# B&R Automation Studio project AutomationsProject
Automation Studio 4.12.6.106; technology packages: mappMotion 5.30.2, mappView 5.24.7

## Configuration Config1

CPU X20CP1382, AutomationRuntime I4.83, Build 4.1.2, Vc V4.73.2

### Task classes (Cpu.sw)
```
Cyclic#4:
  RunBelt <- RunBelt.prg
  main <- main.prg
  ServoTest <- ServoTest.prg
DataObjects: McAcpSys
NcDataObjects: mcdrivelog
Binaries: FWRules, udbdef, TCData, McAcpSim, McAcpDrv, arconfig, User, sysconf, Role, iomap, asfw, ashwac, ashwd, Config_1, arcoal, arsvcreg, arflatprv
Libraries: CppLibs, McBase, MpBase, McAxis, MpAxis, McAcpAx, astime, asieccon, fileio, runtime, powerlnk, asepl, sys_lib
```

### Hardware
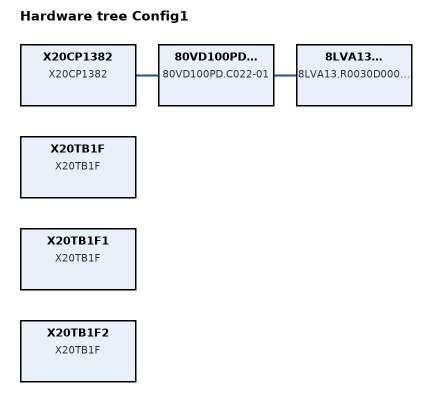
```
80VD100PD.C022-01 : 80VD100PD.C022-01 v2.5.0.0  [PLK1 -> X20CP1382.IF3 (NodeNumber=1) [Cable Type=PowerlinkCable, Length=10, Version=1.0.0.3]; EC1 -> 8LVA13.R0030D000-0.EC]
  DriveConfiguration/Module:
    McAcoposTypeID = AcoposMicroDConfig
    ActivateACOPOSSimulationOnPLC = 0
  DriveConfiguration/Encoder/EncoderX6A/InterfaceType:
    ResolverPolepairs = 1
  DriveConfiguration/Encoder/EncoderX6B/InterfaceType:
    ResolverPolepairs = 1
  DriveConfiguration/Channel[1]/RealAxis:
    AxisReference = FeederAxis
    MechanicalElementsIsInvisible = 0
  DriveConfiguration/Channel[1]/RealAxis/MechanicalElements/Gearbox:
    InputIsReadOnly = 0
    Input = 1
    OutputIsReadOnly = 0
    Output = 1
  DriveConfiguration/Channel[1]/RealAxis/MechanicalElements/RotaryToLinearTransformation:
    ReferenceDistanceIsReadOnly = 0
    ReferenceDistance = 1
  DriveConfiguration/Channel[1]/RealAxis/Controller:
    ModeIsReadOnly = 0
    Mode = PositionController
  DriveConfiguration/Channel[1]/RealAxis/Controller/Mode/Position:
    ProportionalGain = 50
    IntegrationTime = 0.0
    PredictionTime = 0.0004
    TotalDelayTime = 0.0004
  DriveConfiguration/Channel[1]/RealAxis/Controller/Mode/Speed:
    ProportionalGainIsReadOnly = 0
    ProportionalGain = 0.5
    IntegrationTimeIsReadOnly = 0
    IntegrationTime = 0.0
    FilterTimeIsReadOnly = 0
    FilterTime = 0.0
  DriveConfiguration/Channel[1]/RealAxis/Controller/Mode/LoopFilters:
    LoopFilterXIsReadOnly = 0
    LoopFilter1 = NotUsed
    LoopFilter2 = NotUsed
    LoopFilter3 = NotUsed
  DriveConfiguration/Channel[1]/RealAxis/Homing:
    ModeIsReadOnly = 0
    Mode = Direct
  DriveConfiguration/Channel[1]/RealAxis/Homing/Mode:
    Position = 0.0
    ReferencePulse = NotUsed
  DriveConfiguration/Channel[1]/RealAxis/Homing:
    RestorePositionVariable = 
  DriveConfiguration/Channel[1]/RealAxis/StopReaction:
    QuickstopIsReadOnly = 0
    Quickstop = DecelerationLimit
    DriveErrorIsReadOnly = 0
    DriveError = DecelerationLimit
    FilterTime = 0.0
  DriveConfiguration/Channel[1]/RealAxis/MovementErrorLimits:
    PositionError = 1.0
    VelocityErrorMonitoring = NotUsed
  DriveConfiguration/Channel[1]/RealAxis:
    JerkFilterIsReadOnly = 0
    JerkFilter = NotUsed
    ZeroVibrationFilter = NotUsed
  DriveConfiguration/Channel[1]/RealAxis/DigitalInputs/HomingSwitch:
    SourceIsReadOnly = 0
    Source = NotUsed
    Level = High
  DriveConfiguration/Channel[1]/RealAxis/DigitalInputs/PositiveLimitSwitch:
    SourceIsReadOnly = 0
    Source = NotUsed
    Level = High
  DriveConfiguration/Channel[1]/RealAxis/DigitalInputs/NegativeLimitSwitch:
    SourceIsReadOnly = 0
    Source = NotUsed
    Level = High
  DriveConfiguration/Channel[1]/RealAxis/DigitalInputs/Trigger1:
    Source = X2Trigger1
    Level = High
  DriveConfiguration/Channel[1]/RealAxis/DigitalInputs/Trigger2:
    Source = X2Trigger2
    Level = High
  DriveConfiguration/Channel[1]/RealAxis/DigitalInputs/Quickstop:
    Input = Trigger2
  DriveConfiguration/Channel[1]/RealAxis/Simulation:
    SimulationModeOnPLC = SetValueGeneration
    SimulationModeOnACOPOS = NotUsed
  DriveConfiguration/Channel[1]:
    ExternalEncoderAxis = NotUsed
  DriveConfiguration/Channel[2]/RealAxis:
    AxisReference = 
    MechanicalElementsIsInvisible = 0
  DriveConfiguration/Channel[2]/RealAxis/MechanicalElements/Gearbox:
    InputIsReadOnly = 0
    Input = 1
    OutputIsReadOnly = 0
    Output = 1
  DriveConfiguration/Channel[2]/RealAxis/MechanicalElements/RotaryToLinearTransformation:
    ReferenceDistanceIsReadOnly = 0
    ReferenceDistance = 1
  DriveConfiguration/Channel[2]/RealAxis/Controller:
    ModeIsReadOnly = 0
    Mode = PositionController
  DriveConfiguration/Channel[2]/RealAxis/Controller/Mode/Position:
    ProportionalGain = 50.0
    IntegrationTime = 0.0
    PredictionTime = 0.0004
    TotalDelayTime = 0.0004
  DriveConfiguration/Channel[2]/RealAxis/Controller/Mode/Speed:
    ProportionalGainIsReadOnly = 0
    ProportionalGain = 2.0
    IntegrationTimeIsReadOnly = 0
    IntegrationTime = 0.0
    FilterTimeIsReadOnly = 0
    FilterTime = 0.0
  DriveConfiguration/Channel[2]/RealAxis/Controller/Mode/LoopFilters:
    LoopFilterXIsReadOnly = 0
    LoopFilter1 = NotUsed
    LoopFilter2 = NotUsed
    LoopFilter3 = NotUsed
  DriveConfiguration/Channel[2]/RealAxis/Homing:
    ModeIsReadOnly = 0
    Mode = Direct
  DriveConfiguration/Channel[2]/RealAxis/Homing/Mode:
    Position = 0.0
    ReferencePulse = NotUsed
  DriveConfiguration/Channel[2]/RealAxis/Homing:
    RestorePositionVariable = 
  DriveConfiguration/Channel[2]/RealAxis/StopReaction:
    QuickstopIsReadOnly = 0
    Quickstop = DecelerationLimit
    DriveErrorIsReadOnly = 0
    DriveError = DecelerationLimit
    FilterTime = 0.0
  DriveConfiguration/Channel[2]/RealAxis/MovementErrorLimits:
    PositionError = 1.0
    VelocityErrorMonitoring = Automatic1
  DriveConfiguration/Channel[2]/RealAxis:
    JerkFilterIsReadOnly = 0
    JerkFilter = NotUsed
    ZeroVibrationFilter = NotUsed
  DriveConfiguration/Channel[2]/RealAxis/DigitalInputs/HomingSwitch:
    SourceIsReadOnly = 0
    Source = NotUsed
    Level = High
  DriveConfiguration/Channel[2]/RealAxis/DigitalInputs/PositiveLimitSwitch:
    SourceIsReadOnly = 0
    Source = NotUsed
    Level = High
  DriveConfiguration/Channel[2]/RealAxis/DigitalInputs/NegativeLimitSwitch:
    SourceIsReadOnly = 0
    Source = NotUsed
    Level = High
  DriveConfiguration/Channel[2]/RealAxis/DigitalInputs/Trigger1:
    Source = X2Trigger1
    Level = High
  DriveConfiguration/Channel[2]/RealAxis/DigitalInputs/Trigger2:
    Source = X2Trigger2
    Level = High
  DriveConfiguration/Channel[2]/RealAxis/DigitalInputs/Quickstop:
    Input = Trigger2
  DriveConfiguration/Channel[2]/RealAxis/Simulation:
    SimulationModeOnPLC = SetValueGeneration
    SimulationModeOnACOPOS = NotUsed
  DriveConfiguration/Channel[2]:
    ExternalEncoderAxis = NotUsed
8LVA13.R0030D000-0 : 8LVA13.R0030D000-0 v2.2.0.5  [EC -> 80VD100PD.C022-01.EC1; MT -> 80VD100PD.C022-01.MT1]
  M1/MotorParameters:
    MOTOR_AMB_TEMP_RATED = 40
X20CP1382 : X20CP1382 v1.15.0.0  [X1 -> X1.SL; X2 -> X2.SL; X3 -> X3.SL]
  Module X1 (Type=X1, Virtual=true, Version=1.15.0.0)
    Connection (Connector=SS1, TargetModule=X20TB1F, TargetConnector=SS)
    Connection (Connector=SL, TargetModule=X20CP1382, TargetConnector=X1)
    X1AI_ChannelType01 = 4 to 20mA
  Module X2 (Type=X2, Virtual=true, Version=1.15.0.0)
    Connection (Connector=SS1, TargetModule=X20TB1F1, TargetConnector=SS)
    Connection (Connector=SL, TargetModule=X20CP1382, TargetConnector=X2)
  Module X3 (Type=X3, Virtual=true, Version=1.15.0.0)
    Connection (Connector=SS1, TargetModule=X20TB1F2, TargetConnector=SS)
    Connection (Connector=SL, TargetModule=X20CP1382, TargetConnector=X3)
    X3Channel09Source = PWMout
    X3Channel10Source = PWMout
  Connector IF2:
    ActivateDevice = 1
    Mode = Manual
    InternetAddress = 192.168.1.5
    SubnetMask = 255.255.255.0
    InaNodeNumber = 0
  ConfigurationID = testFreq_Config1
  ActivateOpcUa = 1
  OpcUaInformationModels_PV_Version = 1
X20TB1F : X20TB1F v1.0.0.0
X20TB1F1 : X20TB1F v1.0.0.0
X20TB1F2 : X20TB1F v1.0.0.0
```

### IoMap.iom - X20CP1382/IoMap.iom
```iecst
VAR_CONFIG
	::IO_Output.BELT_START AT %QX."X3".DigitalOutput01; (*24 VDC / 0.5 A, source To I1*)
	::IO_Output.BELT_DIR AT %QX."X3".DigitalOutput02; (*24 VDC / 0.5 A, source To I2*)
	::IO_Output.BELT_CONST_SPEED AT %QX."X3".DigitalOutput03; (*24 VDC / 0.5 A, source To I5*)
	::IO_Output._BELT_ACC_ AT %QW."X3".PWMOutput09; (*Pulse width modulation, 24 VDC / 0.2 A [0 to 100.0 %] To I3*)
	::IO_Output._BELT_DEACC_ AT %QW."X3".PWMOutput10; (*Pulse width modulation, 24 VDC / 0.2 A [0 to 100.0 %] To I4*)
	::IO_Output.PWM_PERIOD AT %QW."X3".PWMPeriod09;
	::IO_Output.PWM_PERIOD AT %QW."X3".PWMPeriod10;
	::IO_Input._Distance AT %IW."X1".AnalogInput01;
	::IO_Input.ROBOT_READY AT %IX."X1".DigitalInput01;
	::IO_Output.ROBOT_RUN_PRG AT %QX."X3".DigitalOutput07;
END_VAR
```

### Config_1.axis - X20CP1382/mappMotion/Config_1.axis
```
Element FeederAxis (Type=axis)
  BaseTypeIsReadOnly = 0
  BaseType = Linear
    MeasurementUnit = 5066068
    MeasurementResolutionIsReadOnly = 0
    MeasurementResolution = 0.01
    CountDirectionIsReadOnly = 0
    CountDirection = Standard
  MovementLimitsIsReadOnly = 0
  MovementLimits = Internal
    Position:
      LowerLimitMin = -1.79769313486231E308
      UpperLimitMax = 1.79769313486231E308
      LowerLimit = -1000.0
      UpperLimit = 1000.0
    VelocityIsReadOnly = 0
    Velocity:
      VelocityMax = 3.4E38
      Velocity = 10.0
    AccelerationIsReadOnly = 0
    Acceleration:
      AccelerationMax = 3.4E38
      Acceleration = 50.0
    DecelerationIsReadOnly = 0
    Deceleration:
      DecelerationMax = 3.4E38
      Deceleration = 50.0
  Alarms = None
```

## Logical view

Binary libraries used (declarations not repeated): operator, runtime, astime, AsIecCon, McBase 5.30.2, MpBase, McAxis 5.30.2, MpAxis 5.30.2, McAcpAx 5.30.2

### Global.typ - Global data types
```iecst
TYPE
	ST_Output : 	STRUCT
		PWM_PERIOD : UINT;
		BELT_START : BOOL; (*I1*)
		BELT_DIR : BOOL; (*I2*)
		BELT_CONST_SPEED : BOOL; (*I5*)
		_BELT_DEACC_ : INT; (*I4*)
		_BELT_ACC_ : INT; (*I3*)
		ROBOT_RUN_PRG : BOOL;
	END_STRUCT;
	ST_Input : 	STRUCT
		_Distance : INT; (*Distance sensor on the bottom of the track*)
		ROBOT_READY : BOOL;
		Distance : REAL;
	END_STRUCT;
	packML :
		(
		EXECUTE,
		COMPLETING,
		COMPLETED,
		RESETTING,
		ABORTING,
		ABORTED,
		CLEARING,
		STOPPING,
		STOPPED,
		SUSPENDING,
		SUSPENDED,
		UNSUSPENDING,
		UNHOLDING,
		HELD,
		HOLDING,
		STARTING,
		IDLE
		);
END_TYPE
```

### Global.var - Global variables
```iecst
VAR
	IO_Output : ST_Output;
	IO_Input : ST_Input;
END_VAR
VAR CONSTANT
	ACCEPTED_DISTANCE : REAL := 0.005;
	ROBOT_CATCH_DISTANCE : REAL := 0.22;
END_VAR
```

### Package Logical/Libraries - Global libraries

### Library Logical/Libraries/CppLibs (ANSIC)

#### myStdLib.h
```c
#ifndef MYSTDLIB_H
#define MYSTDLIB_H

#include <stdlib.h>

template<typename T>
inline T abs(T x)
{
	return x < 0 ? -x : x;
}

#endif
```

### Program Logical/main (IEC)

#### Variables.var
```iecst
VAR
	PACK_ML : packML;
	PackMLChar : STRING[80];
END_VAR
```

#### Action.st
```iecst
ACTION States:
	CASE PACK_ML OF
		ABORTING:
			PackMLChar := 'ABORTING';
			PACK_ML := ABORTED;

		ABORTED:
			PackMLChar := 'ABORTED';
			PACK_ML := CLEARING;

		CLEARING:
			PackMLChar := 'CLEARING';
			PACK_ML := STOPPED;

		STOPPING:
			PackMLChar := 'STOPPING';
			PACK_ML := ABORTED;

		STOPPED:
			PackMLChar := 'STOPPED';
			PACK_ML := RESETTING;

		RESETTING:
			PackMLChar := 'RESETTING';
			PACK_ML := IDLE;

		IDLE:
			PackMLChar := 'IDLE';
			PACK_ML := STARTING;

		STARTING:
			PackMLChar := 'STARTING';
			PACK_ML := EXECUTE;

		EXECUTE:
			PackMLChar := 'EXECUTE';
			(*

			The belt should run. If we are in an acceptable region we should go to the position of tray and catch it with the robot.
			This program only tells the robot TO run, not where TO run.

			*)
			IF ACCEPTED_DISTANCE > ABS(ROBOT_CATCH_DISTANCE - IO_Input.Distance) THEN
				IF IO_Input.ROBOT_READY THEN
					IO_Output.BELT_START := FALSE;
					IO_Output.ROBOT_RUN_PRG := TRUE;
				ELSE
					IO_Output.BELT_START := FALSE;
					IO_Output.ROBOT_RUN_PRG := FALSE;
				END_IF
			ELSE
				IO_Output.ROBOT_RUN_PRG := FALSE;

				IF (ROBOT_CATCH_DISTANCE - IO_Input.Distance) > 0 THEN
					IO_Output.BELT_CONST_SPEED := TRUE;
					IO_Output.BELT_DIR := TRUE;
					IO_Output.BELT_START := TRUE;
				ELSE
					IO_Output.BELT_CONST_SPEED := TRUE;
					IO_Output.BELT_DIR := FALSE;
					IO_Output.BELT_START := TRUE;
				END_IF

			END_IF

			//PACK_ML := COMPLETING;
		SUSPENDING:
			PackMLChar := 'SUSPENDING';
			PACK_ML := SUSPENDED;

		SUSPENDED:
			PackMLChar := 'SUSPENDED';
			PACK_ML := UNSUSPENDING;

		UNSUSPENDING:
			PackMLChar := 'UNSUSPENDING';
			PACK_ML := EXECUTE;

		HOLDING:
			PackMLChar := 'HOLDING';
			PACK_ML := HELD;

		HELD:
			PackMLChar := 'HELD';
			PACK_ML := UNHOLDING;

		UNHOLDING:
			PackMLChar := 'UNHOLDING';
			PACK_ML := EXECUTE;

		COMPLETING:
			PackMLChar := 'COMPLETING';
			PACK_ML := COMPLETED;

		COMPLETED:
			PackMLChar := 'COMPLETED';
			PACK_ML := RESETTING;

	END_CASE
END_ACTION
```

#### Main.st
```iecst
PROGRAM _INIT
	(* Insert code here *)

	PACK_ML := CLEARING;

END_PROGRAM

PROGRAM _CYCLIC
	(* Insert code here *)

	IF IO_Input._Distance < 1000 OR IO_Input._Distance > 32000 THEN
		IO_Input.Distance := 1.0;
	ELSE
		IO_Input.Distance := 0.00001033592*IO_Input._Distance+0.1581395;
	END_IF

	States;  // action

	IO_Input.ROBOT_READY; //Kanal 601 - output på robot

	IO_Output.ROBOT_RUN_PRG; //Kanal 501 - input på robot

END_PROGRAM

PROGRAM _EXIT
	(* Insert code here *)

END_PROGRAM
```

### Program Logical/RunBelt (ANSIC)

#### Variables.var
```iecst
VAR
	BELT_SPEED : REAL; (*Belt speed target*)
	_BELT_CURRENT_SPEED_ : REAL; (*Current belt speed*)
	_BELT_ACCELERATION_ : INT; (*Acceleration to belt speed target*)
END_VAR
```

#### Main.cpp
```cpp
#include <bur/plctypes.h>
#ifdef _DEFAULT_INCLUDES
	#include <AsDefault.h>
#endif

#include <cmath>
#include <string>
#include <vector>
#include <map>
#include "../Libraries/CppLibs/myStdLib.h"
//#include <myStdLib.h>

#define INDIFFERENT_SPEED_DIFF 0.5 // [m/s]

std::vector<double> something(50);

// amount of memory to be allocated for heap storage must be specified for every ANSI C++ program with the bur_heap_size variable
unsigned long bur_heap_size = 0xFFFF;

void _INIT ProgramInit(void)
{
	// Insert code here
	double PeriodInHz = 100.0;
	IO_Output.PWM_PERIOD = static_cast<int>((1/PeriodInHz)*1000000);

	IO_Output.BELT_START = true;

	IO_Output.BELT_CONST_SPEED = false; //Hvis du flipper den her, kan du styre hastigheden på inverteren
}

void _CYCLIC ProgramCyclic(void)
{
	// Insert code here
	if( !IO_Output.BELT_CONST_SPEED ) {

		if(BELT_SPEED < 0) {
			IO_Output.BELT_DIR = true;
			IO_Output.BELT_START = true;
		}
		else if(BELT_SPEED > 0) {
			IO_Output.BELT_DIR = false;
			IO_Output.BELT_START = true;
		}
		else {
			IO_Output.BELT_START = false;
		}

		if(fabs(BELT_SPEED - _BELT_CURRENT_SPEED_) > INDIFFERENT_SPEED_DIFF) {

			if(BELT_SPEED < _BELT_CURRENT_SPEED_) {

				_BELT_ACCELERATION_ = -1000;
			}
			else {

				_BELT_ACCELERATION_ = 1000;
			}

		}
		else {

			_BELT_ACCELERATION_ = 0;
		}
	}

	if(_BELT_ACCELERATION_ < 0) {

		IO_Output._BELT_ACC_ = 0;
		IO_Output._BELT_DEACC_ = abs(_BELT_ACCELERATION_);
	} else if(_BELT_ACCELERATION_ > 0) {

		IO_Output._BELT_ACC_ = abs(_BELT_ACCELERATION_);
		IO_Output._BELT_DEACC_ = 0;
	} else {

		IO_Output._BELT_ACC_ = 0;
		IO_Output._BELT_DEACC_ = 0;
	}

}

void _EXIT ProgramExit(void)
{
	// Insert code here

}
```

### Program Logical/ServoTest (IEC)

#### Main.st - Init, cyclic, exit code
```iecst
PROGRAM _INIT
	(* Insert code here *)
	PowerON.Axis := ADR( FeederAxis );
	Home.Axis := ADR ( FeederAxis );
	MoveVelocity.Axis := ADR( FeederAxis );
	StopMotion.Axis := ADR( FeederAxis );
	ResetDrive.Axis := ADR( FeederAxis );

	MoveVelocity.Acceleration := 1.0;
	MoveVelocity.Deceleration := 1.0;

END_PROGRAM

PROGRAM _CYCLIC
	(* Insert code here *)

	(*Feeder.Axis := ADR( FeederAxis );
	Feeder.Enable := TRUE;
	Feeder.Velocity := STRING_TO_REAL( HMI_FeederVelocity );
	Feeder();*)

	IF HMI_Stop AND State = SERVO_MOVE_VEL THEN
		State := SERVO_STOP;
	END_IF

	IF HMI_Reset THEN
		State := SERVO_RESET;
	END_IF

	CASE State OF

		SERVO_IDLE:

			IF HMI_Start THEN
				ServoRun := FALSE;
				State := SERVO_POWER_ON;
			END_IF

		SERVO_POWER_ON:

			PowerON.Enable := TRUE;
			PowerON();

			IF PowerON.Status THEN
				//State := SERVO_MOVE_VEL;
				State := SERVO_HOMING;
			END_IF;

		SERVO_HOMING:

			Home.Position := 0;
			Home.Execute := TRUE;
			Home();

			IF Home.Done THEN
				State := SERVO_MOVE_VEL;
				Home( Execute := FALSE );
			ELSIF Home.Error THEN
				Home( Execute := FALSE );
				State := SERVO_ERROR;
				ErrorState := 'HOME';
			END_IF

		SERVO_MOVE_VEL:

			IF MoveVelocity.Velocity <> STRING_TO_REAL( HMI_FeederVelocity ) THEN
				MoveVelocity.Execute := FALSE;
				MoveVelocity.Velocity := STRING_TO_REAL( HMI_FeederVelocity );
			ELSE
				MoveVelocity.Execute := TRUE;
			END_IF
			IF HMI_FeederDir THEN
				MoveVelocity.Direction := mcDIR_NEGATIVE;
			ELSE
				MoveVelocity.Direction := mcDIR_POSITIVE;
			END_IF
			MoveVelocity();

			IF MoveVelocity.Error THEN
				State := SERVO_ERROR;
				MoveVelocity( Execute := FALSE );
				ErrorState := 'MOVE_VEL';
			END_IF

		SERVO_STOP:

			MoveVelocity( Execute := FALSE );
			StopMotion.Execute := TRUE;
			StopMotion();

			IF StopMotion.Done THEN
				StopMotion( Execute := FALSE );
				State := SERVO_IDLE;
			END_IF

		SERVO_POWER_OFF:

			PowerON( Enable := FALSE );

			IF PowerON.Busy = FALSE THEN
				State := SERVO_IDLE;
			END_IF

		SERVO_RESET:

			MoveVelocity( Execute := FALSE );

			ResetDrive.Execute := TRUE;
			ResetDrive();

			IF ResetDrive.Done THEN
				ResetDrive( Execute := FALSE );
				State := SERVO_POWER_OFF;
			END_IF

		SERVO_ERROR:

			IF ResetServo THEN
				ResetServo := FALSE;
				State := SERVO_RESET;
				ErrorState := '';
			END_IF

	END_CASE

END_PROGRAM

PROGRAM _EXIT
	(* Insert code here *)

END_PROGRAM
```

#### Types.typ - Local data types
```iecst
TYPE
	E_ServoStates :
		(
		SERVO_IDLE,
		SERVO_POWER_ON,
		SERVO_MOVE_VEL,
		SERVO_RESET,
		SERVO_STOP,
		SERVO_POWER_OFF,
		SERVO_ERROR,
		SERVO_HOMING,
		SERVO_OFF
		);
END_TYPE
```

#### Variables.var - Local variables
```iecst
VAR
	PowerON : MC_Power;
	HMI_FeederVelocity : STRING[80];
	State : E_ServoStates;
	MoveVelocity : MC_MoveVelocity;
	ServoRun : BOOL;
	StopMotion : MC_Stop;
	ResetDrive : MC_Reset;
	Home : MC_Home;
	TestVelocity : REAL := 100.0;
	ResetServo : BOOL;
	ErrorState : STRING[80];
	Feeder : FB_ServoControl;
	HMI_Stop : BOOL;
	HMI_Reset : BOOL;
	HMI_Start : BOOL;
	HMI_FeederDir : BOOL;
END_VAR
```

#### LocalFunctions.fun
```iecst
{REDUND_ERROR} FUNCTION_BLOCK FB_ServoControl (*TODO: Add your comment here*) (*$GROUP=User,$CAT=User,$GROUPICON=User.png,$CATICON=User.png*)
	VAR_INPUT
		Axis : REFERENCE TO McAxisType;
		Enable : BOOL;
		Stop : BOOL;
		Reset : BOOL;
		Velocity : REAL;
		Acc : REAL := 1.0;
		Dec : REAL := 1.0;
	END_VAR
	VAR_OUTPUT
		Error : BOOL;
		ErrorCode : INT;
		isRunning : BOOL;
	END_VAR
	VAR
		McPower : MC_Power;
		McHome : MC_Home;
		McStop : MC_Stop;
		McReset : MC_Reset;
		McMoveVel : MC_MoveVelocity;
		State : E_ServoStates := SERVO_OFF;
	END_VAR
END_FUNCTION_BLOCK
```

#### FB_ServoControl.st
```iecst
(* TODO: Add your comment here *)
FUNCTION_BLOCK FB_ServoControl

	McPower.Axis	:= ADR( Axis );
	McHome.Axis 	:= ADR( Axis );
	McMoveVel.Axis 	:= ADR( Axis );
	McStop.Axis 	:= ADR( Axis );
	McReset.Axis 	:= ADR( Axis );

	McMoveVel.Acceleration := Acc;
	McMoveVel.Deceleration := Dec;

	IF NOT Enable AND isRunning THEN
		State := SERVO_POWER_OFF;
	ELSIF NOT Enable THEN
		State := SERVO_IDLE;
	ELSIF Stop AND isRunning THEN
		State := SERVO_STOP;
	END_IF

	CASE State OF

		SERVO_OFF:

			ErrorCode := 0;

			IF Enable THEN
				isRunning := TRUE;
				State := SERVO_POWER_ON;
			END_IF

		SERVO_IDLE:

			ErrorCode := 0;

		SERVO_POWER_ON:

			McPower.Enable := TRUE;

			IF McPower.Status THEN
				State := SERVO_HOMING;
			END_IF;

			McPower();

		SERVO_HOMING:

			McHome.Position := 0;
			McHome.Execute := TRUE;

			IF McHome.Done THEN
				State := SERVO_MOVE_VEL;
				McHome.Execute := FALSE;
			ELSIF McHome.Error THEN
				McHome.Execute := FALSE;
				State := SERVO_ERROR;
				ErrorCode := 1001;
			END_IF

			McHome();

		SERVO_MOVE_VEL:

			McMoveVel.Velocity := Velocity;
			McMoveVel.Execute := TRUE;

			IF McMoveVel.Error THEN
				State := SERVO_ERROR;
				McMoveVel.Execute := FALSE;
				ErrorCode := 2001;
			END_IF

			McMoveVel();

		SERVO_STOP:

			McMoveVel.Execute := FALSE;
			McStop.Execute := TRUE;

			IF McStop.Done THEN
				isRunning := FALSE;
				McStop.Execute := FALSE;
				State := SERVO_IDLE;
			END_IF

			McStop();

		SERVO_POWER_OFF:

			McPower.Enable := FALSE;

			IF McPower.Busy = FALSE THEN
				State := SERVO_OFF;
			END_IF

			McPower();

		SERVO_RESET:

			McReset.Execute := TRUE;

			IF McReset.Done THEN
				McReset.Execute := FALSE;
				State := SERVO_IDLE;
			END_IF

			McReset();

		SERVO_ERROR:

			isRunning := FALSE;

			IF Reset THEN
				State := SERVO_RESET;
			END_IF

	END_CASE

END_FUNCTION_BLOCK
```

- Visualisation Logical/mappView (not shown)

### Program Logical/packML

#### Main.st
```iecst
PROGRAM _INIT
	(* Insert code here *)

	PACK_ML := CLEARING;

END_PROGRAM

PROGRAM _CYCLIC
	(* Insert code here *)
	CASE PACK_ML OF
		ABORTING:
			PACK_ML := ABORTED;
		ABORTED:
			PACK_ML := CLEARING;
		CLEARING:
			PACK_ML := STOPPED;
		STOPPING:
			PACK_ML := ABORTED;
		STOPPED:
			PACK_ML := RESETTING;
		RESETTING:
			PACK_ML := IDLE;
		IDLE:
			PACK_ML := STARTING;
		STARTING:
			PACK_ML := EXECUTE;
		EXECUTE:
			//PACK_ML := COMPLETING;
		SUSPENDING:
			PACK_ML := SUSPENDED;
		SUSPENDED:
			PACK_ML := UNSUSPENDING;
		UNSUSPENDING:
			PACK_ML := EXECUTE;
		HOLDING:
			PACK_ML := HELD;
		HELD:
			PACK_ML := UNHOLDING;
		UNHOLDING:
			PACK_ML := EXECUTE;
		COMPLETING:
			PACK_ML := COMPLETED;
		COMPLETED:
			PACK_ML := RESETTING;
		END_CASE
END_PROGRAM

PROGRAM _EXIT
	(* Insert code here *)

END_PROGRAM
```

### Program Logical/Program

#### Variables.var
```iecst
VAR
	BELT_START : BOOL; (*I1*)
	BELT_DIR : BOOL; (*I2*)
	BELT_CONST_SPEED : BOOL; (*I5*)
	BELT_SPEED : REAL; (*Belt speed target*)
	_BELT_CURRENT_SPEED_ : REAL; (*Current belt speed*)
	_BELT_ACCELERATION_ : INT; (*Acceleration to belt speed target*)
	_BELT_DEACC_ : INT; (*I4*)
	_BELT_ACC_ : INT; (*I3*)
END_VAR
```

#### Main.cpp
```cpp
#include <bur/plctypes.h>

#ifdef _DEFAULT_INCLUDES
	#include <AsDefault.h>
#endif

// amount of memory to be allocated for heap storage must be specified for every ANSI C++ program with the bur_heap_size variable
unsigned long bur_heap_size = 0xFFFF;

void _INIT ProgramInit(void)
{
	// Insert code here
	PeriodInHz = 100;
	PWM_PERIOD = (1/PeriodInHz)*1000000;

}

void _CYCLIC ProgramCyclic(void)
{
	// Insert code here

}

void _EXIT ProgramExit(void)
{
	// Insert code here

}
```
